(* Schneider Machine Expert - Basic project multiple timers, file version 2.0.0.0 *)
(* ProjectInformations: Name=New project *)

HARDWARE
  Cpu 0: TM221CE16R
  EthernetConfiguration: NetworkName=M221, IpAllocationMode=FixedAddress, IpAddress=0.0.0.0, SubnetMask=0.0.0.0
  SerialLineConfiguration: Baud=Baud19200, Parity=ParityEven, DataBits=DataBits8, StopBits=StopBits1, PhysicalMedium=PhysicalMediumRs485, TransmissionMode=TransmissionModeModbusRtu, SlaveId=1, Addressing=SlaveAddressing
  MastTask: UsePeriodScanMode=false, PeriodScan=100
  FastTask: Period=255
  CpuBehavior: StartingMode=StartAsPreviousState, AutoSaveRamOnEeprom=true, WatchdogPeriod=250

SYMBOLS  (address, symbol, comment, settings)

POU New POU
  (* SectionNumber=0 *)

// Rung 0
  BLK %TM0
  LD %I0.0
  IN
  OUT_BLK
  LD Q
  ST %Q0.0
  END_BLK
  // as ST:
  //   %TM0(IN := %I0.0);
  //   %Q0.0 := %TM0.Q;

// Rung 1
  BLK %TM1
  LD %I0.0
  IN
  OUT_BLK
  LD Q
  ST %Q0.1
  END_BLK
  // as ST:
  //   %TM1(IN := %I0.0);
  //   %Q0.1 := %TM1.Q;

// Rung 2
  BLK %TM2
  LD %I0.0
  IN
  OUT_BLK
  LD Q
  ST %Q0.2
  END_BLK
  // as ST:
  //   %TM2(IN := %I0.0);
  //   %Q0.2 := %TM2.Q;

// Rung 3
  BLK %TM3
  LD %I0.0
  IN
  OUT_BLK
  LD Q
  ST %Q0.3
  END_BLK
  // as ST:
  //   %TM3(IN := %I0.0);
  //   %Q0.3 := %TM3.Q;

// Rung 4
  BLK %TM4
  LD %I0.0
  IN
  OUT_BLK
  LD Q
  ST %Q0.6
  END_BLK
  // as ST:
  //   %TM4(IN := %I0.0);
  //   %Q0.6 := %TM4.Q;

// Rung 5
  BLK %TM5
  LD %I0.0
  IN
  OUT_BLK
  LD Q
  ST %Q0.4
  END_BLK
  // as ST:
  //   %TM5(IN := %I0.0);
  //   %Q0.4 := %TM5.Q;

// Rung 6
  BLK %TM6
  LD %I0.0
  IN
  OUT_BLK
  LD Q
  ST %Q0.5
  END_BLK
  // as ST:
  //   %TM6(IN := %I0.0);
  //   %Q0.5 := %TM6.Q;

// Rung 7
  BLK %TM7
  LD %I0.0
  IN
  OUT_BLK
  LD Q
  ST %M0
  END_BLK
  // as ST:
  //   %TM7(IN := %I0.0);
  //   %M0 := %TM7.Q;

// Rung 8
  BLK %TM8
  LD %I0.0
  IN
  OUT_BLK
  LD Q
  ST %M2
  END_BLK
  // as ST:
  //   %TM8(IN := %I0.0);
  //   %M2 := %TM8.Q;

// Rung 9
  BLK %TM9
  LD %I0.0
  IN
  OUT_BLK
  LD Q
  ST %M3
  END_BLK
  // as ST:
  //   %TM9(IN := %I0.0);
  //   %M3 := %TM9.Q;

// Rung 10
  BLK %TM10
  LD %I0.0
  IN
  OUT_BLK
  LD Q
  ST %M3
  END_BLK
  // as ST:
  //   %TM10(IN := %I0.0);
  //   %M3 := %TM10.Q;

// Rung 11
  BLK %TM11
  LD %I0.0
  IN
  OUT_BLK
  LD Q
  ST %M3
  END_BLK
  // as ST:
  //   %TM11(IN := %I0.0);
  //   %M3 := %TM11.Q;

// Rung 12
  BLK %TM12
  LD %I0.0
  IN
  OUT_BLK
  LD Q
  ST %M3
  END_BLK
  // as ST:
  //   %TM12(IN := %I0.0);
  //   %M3 := %TM12.Q;

// Rung 13
  BLK %TM13
  LD %I0.0
  IN
  OUT_BLK
  LD Q
  ST %M3
  END_BLK
  // as ST:
  //   %TM13(IN := %I0.0);
  //   %M3 := %TM13.Q;

// Rung 14
  BLK %TM14
  LD %I0.0
  IN
  OUT_BLK
  LD Q
  ST %M3
  END_BLK
  // as ST:
  //   %TM14(IN := %I0.0);
  //   %M3 := %TM14.Q;

// Rung 15
  BLK %TM15
  LD %I0.0
  IN
  OUT_BLK
  LD Q
  ST %M3
  END_BLK
  // as ST:
  //   %TM15(IN := %I0.0);
  //   %M3 := %TM15.Q;
